{attribute 'linkalways'} 
{attribute 'no_explicit_call' := 'This FB is a CLASS and must be accessed using methods or properties'}
{attribute 'enable_dynamic_creation'}
FUNCTION_BLOCK PUBLIC ABSTRACT BaseMotionCommand EXTENDS NoopAsyncCommand IMPLEMENTS MotionCommand
VAR
END_VAR

{attribute 'monitoring' := 'call'}
PROPERTY PUBLIC ABSTRACT Active : BOOL
GET // PUBLIC
END_GET
END_PROPERTY

METHOD PROTECTED ABSTRACT OnExecuting
VAR_INPUT
	state_control : AsyncCommandStateControl;
END_VAR
END_METHOD

END_FUNCTION_BLOCK

(* stored: Version 1.1.0.1
   POU BaseMotionCommand: Id {031054ba-f892-0de3-09de-fc1b37e54d8c}, SpecialFunc None
   Property Active: Id {6e440f34-2bfa-01bb-08ff-9edd6af43fbb}
   Get Get: Id {f0c67215-0008-0488-0c4d-4470e62a6019}
   Method OnExecuting: Id {0faeb363-a03a-046b-0514-184c987e2eaa} *)
